(* CODESYS project 4b.project

Project tree, tasks and I/O mapping:
  Device : CODESYS Control Win V3, 3S - Smart Software Solutions GmbH, order no. 305021, version 3.5.11.30
    application Application
      libraries: Standard, * (System)
      task MainTask (cyclic, interval t#20ms, priority 1) calls PLC_PRG
      program PLC_PRG [LD]
*)

// Device/Application/PLC_PRG
PROGRAM PLC_PRG
VAR
	KM1: BOOL;
	SB2: BOOL;
	FR: BOOL;
	SB1: BOOL;
	KM2: BOOL;
	SB3: BOOL;
	H1: BOOL;
	H2: BOOL;
	H3: BOOL;
END_VAR

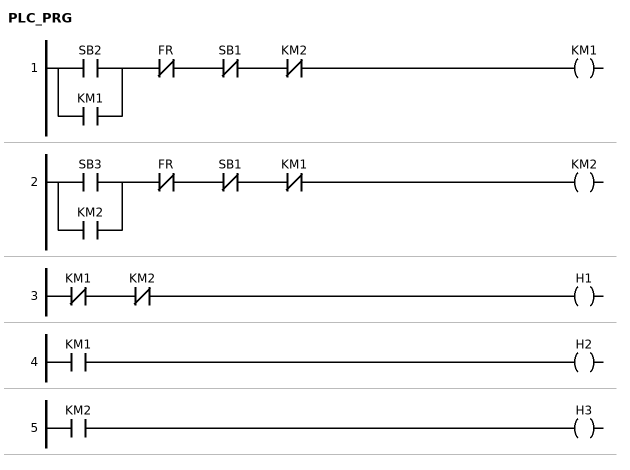
// NETWORK 1
KM1 := (SB2 OR KM1) AND NOT FR AND NOT SB1 AND NOT KM2;

// NETWORK 2
KM2 := (SB3 OR KM2) AND NOT FR AND NOT SB1 AND NOT KM1;

// NETWORK 3
H1 := NOT KM1 AND NOT KM2;

// NETWORK 4
H2 := KM1;

// NETWORK 5
H3 := KM2;

END_PROGRAM
